ABB RobotStudio station: zaliczenie_zadanie1_20200109-012039.rsstn

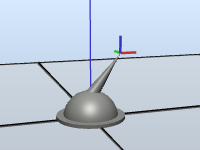
Station zaliczenie_zadanie1 (saved by RobotStudio 6.8.8307.1040)
Controller IRB_6640_185kg_2.80m
  mechanical unit ROB_1: IRB6640_185_280__04, 6 joints, base frame (0, 0, 0) mm
Layout (positions relative to the parent item):
  - IRB6640_185_280__04 [mechanism, from Robots\IRB6640_185_280_G_04.rslib] at (0, 0, 0) mm; joint values [0, 0, 0, 0, 0.5236, 0] (rad or m)
  - bolec [mechanism] at (0, 0, 0) mm
      TCP bolec at (90.27, 0, 185) mm
      links: Part_12
